DATA_BLOCK "AutoProcessData_Buffer_Clear"
VAR
  DataBuffer : Array[0..60] of "ProcessData";
  DataBufferClear : "ProcessData";
  VAL : Int;
END_VAR
BEGIN
END_DATA_BLOCK
